TEXTLIST TextList_ISSerrorid
  0 = 'no_error'
  1 = 'not_connected'
  2 = 'invalid_state'
  4 = 'pump1_failure'
  6 = 'pump2_failure'
  7 = 'time_out'
  8 = 'back_to_air_tank'
  9 = 'io_error'
  10 = 'unknown_error'
  666 = 'emergency_error'
   = ''
END_TEXTLIST

(* stored: Version 1.1.0.1, ProductVersion 3.1.4024.11
   TextList TextList_ISSerrorid: Id {2532d1fd-e8e7-472d-8ac1-1d1ee19c9b52} *)
